(* IEC 61131-3 sources: codesys_template_public/codesys_export/Device/Application/Function Blocks/MC_BasicControl, 26 files *)

(* ---- MC_ActualDriver_SetPosition.st ---- *)
// X57s 驅動器不支援標準 MC_SetPosition（Set Position 指令）
// 使用 Homing Mode 35 模擬 SetPosition 的功能作為 Workaround
FUNCTION_BLOCK MC_ActualDriver_SetPosition
VAR_IN_OUT
	Axis : AXIS_REF_SM3;
END_VAR
VAR_INPUT
	Execute		: BOOL;
	Position	: LREAL;
	xReset		: BOOL;
END_VAR
VAR_OUTPUT
	Done	: BOOL;
	Busy	: BOOL;
	Error	: BOOL;
	ErrorID	: SM3_Basic.SMC_ERROR;
END_VAR
VAR
	iStep : INT;
	_fbMC_WriteHomingParameters : MC_WriteHomingParameters;
	_stFakeHomingParameter : structAxisControl_HomingProfile := (uiHomingMethod := 35);
	_fbMC_Home : MC_Home;
END_VAR

// === IMPLEMENTATION ===
_fbMC_WriteHomingParameters(Axis := Axis, xEnable := TRUE, stParameter := _stFakeHomingParameter);
_fbMC_Home(Axis := Axis, Position := Position);

CASE iStep OF
	0: // 等待 Execute
	_fbMC_WriteHomingParameters.xExecute := FALSE;
	_fbMC_Home.Execute := FALSE;
	Done := FALSE;
	Error := FALSE;
	Busy := FALSE;
	IF Execute THEN
		iStep := iStep + 1;
	END_IF

	1: // 寫入 Homing 參數（Homing Mode 35）
	_fbMC_WriteHomingParameters.xExecute := TRUE;
	Busy := TRUE;
	IF _fbMC_WriteHomingParameters.xDone THEN
		_fbMC_WriteHomingParameters.xExecute := FALSE;
		iStep := iStep + 1;
	END_IF
	IF _fbMC_WriteHomingParameters.xError THEN
		Error := TRUE;
		iStep := 9999;
	END_IF

	2: // 執行 MC_Home（使用 Mode 35 觸發位置設定）
	_fbMC_Home.Execute := TRUE;
	IF _fbMC_Home.Done THEN
		_fbMC_Home.Execute := FALSE;
		iStep := iStep + 1;
	END_IF
	IF _fbMC_Home.Error THEN
		Error := TRUE;
		ErrorID := _fbMC_Home.ErrorID;
		iStep := 9999;
	END_IF

ELSE // iStep >= 3 or 9999
	Done := (iStep <> 9999);
	IF NOT Execute THEN
		iStep := 0;
		Done := FALSE;
		Error := FALSE;
		ErrorID := 0;
	END_IF
END_CASE

IF xReset THEN
	iStep := 0;
	Done := FALSE;
	Error := FALSE;
	ErrorID := 0;
END_IF

(* ---- MC_BasicControl.st ---- *)
FUNCTION_BLOCK ABSTRACT MC_BasicControl EXTENDS BaseStateMachine
VAR_IN_OUT
	Axis        : AXIS_REF_SM3;
	stParameter : structAxisControl_Parameter;
END_VAR
VAR_INPUT
	xEMS         : BOOL;	// 緊急停止（立即，不等減速）
	xJogPositive : BOOL;	// Jog 正方向（跨任務持久訊號，HMI 用）
	xJogNegative : BOOL;	// Jog 負方向（跨任務持久訊號，HMI 用）
END_VAR
VAR_OUTPUT
	xAxisStandStill       : BOOL;	// 軸停止不動
	xPositiveLimitReached : BOOL;	// 正向極限觸動
	xNegativeLimitReached : BOOL;	// 負向極限觸動
	xInVelocity           : BOOL;	// 速度命令中（已達目標速度）
END_VAR
VAR
	// 電源控制旗標（由狀態機與 Stop() 管理）
	_xPowerOn : BOOL;

	// 驅動器 IO 旗標（由 ReadDriverInputs 填入）
	_xPositiveLimitInput : BOOL;
	_xNegativeLimitInput : BOOL;
	_xBrakeInput         : BOOL;
	_wDriverErrorCode    : WORD;

	// 命令請求旗標（當前掃描，由 method 設定）
	_xJogPosRequested  : BOOL;
	_xJogNegRequested  : BOOL;
	_xMoveAbsRequested : BOOL;
	_xMoveRelRequested : BOOL;
	_xMoveVelRequested : BOOL;
	_xHomeRequested    : BOOL;
	_xSetPosRequested  : BOOL;

	// 命令請求旗標（前一掃描，供狀態機讀取）
	_xJogPosRequested_Prev  : BOOL;
	_xJogNegRequested_Prev  : BOOL;
	_xMoveAbsRequested_Prev : BOOL;
	_xMoveRelRequested_Prev : BOOL;
	_xMoveVelRequested_Prev : BOOL;
	_xHomeRequested_Prev    : BOOL;
	_xSetPosRequested_Prev  : BOOL;

	// 命令參數（由 method 解析後填入）
	_lrJogVelocity : LREAL;
	_lrJogAcc      : LREAL;
	_lrJogDec      : LREAL;
	_lrJogJerk     : LREAL;

	_lrSetPosTarget : LREAL;

	// 命令完成追蹤
	_xCommandDone      : BOOL;
	_iActiveCommand    : INT;					// 最近完成的命令對應的 enumAxisControl_Step
	_eLastMotionError  : SM3_Error.SMC_ERROR;	// 最近一次 SM3 動作錯誤碼（供 method 回傳）

	// MoveRelative 重新觸發鎖：Done 後設 TRUE，呼叫端停止呼叫後清除
	// 防止持續呼叫 MoveRelative() 時完成後立刻開始下一次相對移動
	_xMoveRelNeedsReArm : BOOL;

	// 重置後返回步驟
	_iStepBeforeReset : INT;

	// SM3 Motion FBs
	_fbMC_Power                 : MC_Power;
	_fbMC_Reset                 : MC_Reset;
	_fbMC_MoveAbsolute          : MC_MoveAbsolute;
	_fbMC_MoveRelative          : MC_MoveRelative;
	_fbMC_MoveVelocity          : MC_MoveVelocity;
	_fbMC_Stop                  : MC_Stop;
	_fbMC_Stop_EMS              : MC_Stop;
	_fbMC_Home                  : MC_Home;
	_fbMC_WriteHomingParameters : MC_WriteHomingParameters;

	// Jog 速度變化偵測（ContinuousUpdate 邏輯）
	_fbVCD_Jog : ValueChangeDetector;
END_VAR

// === IMPLEMENTATION ===
xEnabled        := Axis.bRegulatorOn;
SUPER^();
_RunMotionFBs();

(* ---- MC_BasicControl_LC10E.st ---- *)
FUNCTION_BLOCK MC_BasicControl_LC10E EXTENDS MC_BasicControl
VAR_INPUT
	wDriverInputWord : WORD;	// X57s PDO 輸入字（位元映射見 ReadDriverInputs）
	wDriverErrorCode : WORD;	// X57s 錯誤碼（PDO 讀取）
END_VAR
VAR
	_fbSetPosition_ActualDriver : MC_ActualDriver_SetPosition;	// Homing Mode 35 workaround
	_xSetPosFirstCall   : BOOL := TRUE;			// 確保 Execute 有上升沿
END_VAR

// === IMPLEMENTATION ===
SUPER^(Axis := Axis, stParameter := stParameter);

(* ---- MC_BasicControl_VisuWrapper.st ---- *)
FUNCTION_BLOCK MC_BasicControl_VisuWrapper
VAR_IN_OUT
	fbAxis   : MC_BasicControl_LC10E;
	stCmd    : structMC_BasicControl_VisuCmd;
	stStatus : structMC_BasicControl_VisuStatus;
END_VAR
VAR
	_xClearLastResultPrev : BOOL;
	_xHomePrev            : BOOL;
	_xResetPrev           : BOOL;
	_xStopPrev            : BOOL;
	_xMoveAbsPrev         : BOOL;
	_xMoveRelPosPrev      : BOOL;
	_xMoveRelNegPrev      : BOOL;
	_xMoveVelPrev         : BOOL;
	_xSetPositionPrev     : BOOL;
	_xHomeLatched         : BOOL;
	_xMoveAbsLatched      : BOOL;
	_xMoveRelLatched      : BOOL;
	_xMoveVelLatched      : BOOL;
	_xSetPositionLatched  : BOOL;
	_udiLastPulseSeq   : UDINT;
END_VAR

// === IMPLEMENTATION ===
// Reject code:
// 1 = NONE command
// 2 = Unknown command
// 3 = Invalid motion parameter
stStatus.xPulseAccepted := FALSE;
stStatus.xPulseRejected := FALSE;
stStatus.iPulseRejectCode := 0;
stStatus.xJogCommanded := FALSE;

IF stCmd.xClearLastResult AND NOT _xClearLastResultPrev THEN
	Clear(stStatus.stLastResult);
END_IF

IF stCmd.xStop AND NOT _xStopPrev THEN
	fbAxis.Stop();
	_xHomeLatched := FALSE;
	_xMoveAbsLatched := FALSE;
	_xMoveRelLatched := FALSE;
	_xMoveVelLatched := FALSE;
	_xSetPositionLatched := FALSE;
	stStatus.xPulseAccepted := TRUE;
END_IF

IF stCmd.xReset AND NOT _xResetPrev THEN
	fbAxis.Reset();
	_xHomeLatched := FALSE;
	_xMoveAbsLatched := FALSE;
	_xMoveRelLatched := FALSE;
	_xMoveVelLatched := FALSE;
	_xSetPositionLatched := FALSE;
	stStatus.xPulseAccepted := TRUE;
END_IF

IF stCmd.udiPulseSeq <> _udiLastPulseSeq THEN
	CASE stCmd.ePulseCmd OF
		enumMC_BasicControl_VisuPulseCmd.STOP:
			fbAxis.Stop();
			_xHomeLatched := FALSE;
			_xMoveAbsLatched := FALSE;
			_xMoveRelLatched := FALSE;
			_xMoveVelLatched := FALSE;
			_xSetPositionLatched := FALSE;
			stStatus.xPulseAccepted := TRUE;
		enumMC_BasicControl_VisuPulseCmd.RESET:
			fbAxis.Reset();
			_xHomeLatched := FALSE;
			_xMoveAbsLatched := FALSE;
			_xMoveRelLatched := FALSE;
			_xMoveVelLatched := FALSE;
			_xSetPositionLatched := FALSE;
			stStatus.xPulseAccepted := TRUE;
		enumMC_BasicControl_VisuPulseCmd.HOME:
			_xHomeLatched := TRUE;
			_xMoveAbsLatched := FALSE;
			_xMoveRelLatched := FALSE;
			_xMoveVelLatched := FALSE;
			_xSetPositionLatched := FALSE;
			stStatus.xPulseAccepted := TRUE;
		enumMC_BasicControl_VisuPulseCmd.MOVE_ABSOLUTE:
			IF stCmd.lrMoveAbsVel < 0.0 OR stCmd.lrMoveAbsAcc < 0.0 OR stCmd.lrMoveAbsDec < 0.0 OR stCmd.lrMoveAbsJerk < 0.0 THEN
				stStatus.xPulseRejected := TRUE;
				stStatus.iPulseRejectCode := 3;
			ELSE
				_xHomeLatched := FALSE;
				_xMoveAbsLatched := TRUE;
				_xMoveRelLatched := FALSE;
				_xMoveVelLatched := FALSE;
				_xSetPositionLatched := FALSE;
				stStatus.xPulseAccepted := TRUE;
			END_IF
		enumMC_BasicControl_VisuPulseCmd.MOVE_RELATIVE:
			IF stCmd.lrMoveRelVel < 0.0 OR stCmd.lrMoveRelAcc < 0.0 OR stCmd.lrMoveRelDec < 0.0 OR stCmd.lrMoveRelJerk < 0.0 THEN
				stStatus.xPulseRejected := TRUE;
				stStatus.iPulseRejectCode := 3;
			ELSE
				_xHomeLatched := FALSE;
				_xMoveAbsLatched := FALSE;
				_xMoveRelLatched := TRUE;
				_xMoveVelLatched := FALSE;
				_xSetPositionLatched := FALSE;
				stStatus.xPulseAccepted := TRUE;
			END_IF
		enumMC_BasicControl_VisuPulseCmd.MOVE_VELOCITY:
			IF stCmd.lrMoveVelAcc < 0.0 OR stCmd.lrMoveVelDec < 0.0 OR stCmd.lrMoveVelJerk < 0.0 THEN
				stStatus.xPulseRejected := TRUE;
				stStatus.iPulseRejectCode := 3;
			ELSE
				_xHomeLatched := FALSE;
				_xMoveAbsLatched := FALSE;
				_xMoveRelLatched := FALSE;
				_xMoveVelLatched := TRUE;
				_xSetPositionLatched := FALSE;
				stStatus.xPulseAccepted := TRUE;
			END_IF
		enumMC_BasicControl_VisuPulseCmd.SET_POSITION:
			_xHomeLatched := FALSE;
			_xMoveAbsLatched := FALSE;
			_xMoveRelLatched := FALSE;
			_xMoveVelLatched := FALSE;
			_xSetPositionLatched := TRUE;
			stStatus.xPulseAccepted := TRUE;
		enumMC_BasicControl_VisuPulseCmd.NONE:
			stStatus.xPulseRejected := TRUE;
			stStatus.iPulseRejectCode := 1;
	ELSE
		stStatus.xPulseRejected := TRUE;
		stStatus.iPulseRejectCode := 2;
	END_CASE

	_udiLastPulseSeq      := stCmd.udiPulseSeq;
	stStatus.udiPulseAckSeq := stCmd.udiPulseSeq;
	stStatus.ePulseAckCmd   := stCmd.ePulseCmd;
END_IF

// Button pulse compatibility path for visu widgets.
IF stCmd.xHome AND NOT _xHomePrev THEN
	_xHomeLatched := TRUE;
	_xMoveAbsLatched := FALSE;
	_xMoveRelLatched := FALSE;
	_xMoveVelLatched := FALSE;
	_xSetPositionLatched := FALSE;
	stStatus.xPulseAccepted := TRUE;
ELSIF stCmd.xMoveAbsoluteExecute AND NOT _xMoveAbsPrev THEN
	IF stCmd.lrMoveAbsVel < 0.0 OR stCmd.lrMoveAbsAcc < 0.0 OR stCmd.lrMoveAbsDec < 0.0 OR stCmd.lrMoveAbsJerk < 0.0 THEN
		stStatus.xPulseRejected := TRUE;
		stStatus.iPulseRejectCode := 3;
	ELSE
		_xHomeLatched := FALSE;
		_xMoveAbsLatched := TRUE;
		_xMoveRelLatched := FALSE;
		_xMoveVelLatched := FALSE;
		_xSetPositionLatched := FALSE;
		stStatus.xPulseAccepted := TRUE;
	END_IF
ELSIF stCmd.xMoveRelativePosExecute AND NOT _xMoveRelPosPrev THEN
	IF stCmd.lrMoveRelVel < 0.0 OR stCmd.lrMoveRelAcc < 0.0 OR stCmd.lrMoveRelDec < 0.0 OR stCmd.lrMoveRelJerk < 0.0 THEN
		stStatus.xPulseRejected := TRUE;
		stStatus.iPulseRejectCode := 3;
	ELSE
		stCmd.lrMoveRelDist := ABS(stCmd.lrMoveRelDist);
		_xHomeLatched := FALSE;
		_xMoveAbsLatched := FALSE;
		_xMoveRelLatched := TRUE;
		_xMoveVelLatched := FALSE;
		_xSetPositionLatched := FALSE;
		stStatus.xPulseAccepted := TRUE;
	END_IF
ELSIF stCmd.xMoveRelativeNegExecute AND NOT _xMoveRelNegPrev THEN
	IF stCmd.lrMoveRelVel < 0.0 OR stCmd.lrMoveRelAcc < 0.0 OR stCmd.lrMoveRelDec < 0.0 OR stCmd.lrMoveRelJerk < 0.0 THEN
		stStatus.xPulseRejected := TRUE;
		stStatus.iPulseRejectCode := 3;
	ELSE
		stCmd.lrMoveRelDist := -ABS(stCmd.lrMoveRelDist);
		_xHomeLatched := FALSE;
		_xMoveAbsLatched := FALSE;
		_xMoveRelLatched := TRUE;
		_xMoveVelLatched := FALSE;
		_xSetPositionLatched := FALSE;
		stStatus.xPulseAccepted := TRUE;
	END_IF
ELSIF stCmd.xMoveVelocityExecute AND NOT _xMoveVelPrev THEN
	IF stCmd.lrMoveVelAcc < 0.0 OR stCmd.lrMoveVelDec < 0.0 OR stCmd.lrMoveVelJerk < 0.0 THEN
		stStatus.xPulseRejected := TRUE;
		stStatus.iPulseRejectCode := 3;
	ELSE
		_xHomeLatched := FALSE;
		_xMoveAbsLatched := FALSE;
		_xMoveRelLatched := FALSE;
		_xMoveVelLatched := TRUE;
		_xSetPositionLatched := FALSE;
		stStatus.xPulseAccepted := TRUE;
	END_IF
ELSIF stCmd.xSetPosition AND NOT _xSetPositionPrev THEN
	_xHomeLatched := FALSE;
	_xMoveAbsLatched := FALSE;
	_xMoveRelLatched := FALSE;
	_xMoveVelLatched := FALSE;
	_xSetPositionLatched := TRUE;
	stStatus.xPulseAccepted := TRUE;
END_IF

IF _xHomeLatched THEN
	stStatus.stLastResult := fbAxis.Home();
	IF stStatus.stLastResult.xDone OR stStatus.stLastResult.xError THEN
		_xHomeLatched := FALSE;
	END_IF
ELSIF _xMoveAbsLatched THEN
	stStatus.stLastResult := fbAxis.MoveAbsolute(
		lrPosition := stCmd.lrMoveAbsPos,
		lrVelocity := stCmd.lrMoveAbsVel,
		lrAcceleration := stCmd.lrMoveAbsAcc,
		lrDeceleration := stCmd.lrMoveAbsDec,
		lrJerk := stCmd.lrMoveAbsJerk
	);
	IF stStatus.stLastResult.xDone OR stStatus.stLastResult.xError THEN
		_xMoveAbsLatched := FALSE;
	END_IF
ELSIF _xMoveRelLatched THEN
	stStatus.stLastResult := fbAxis.MoveRelative(
		lrDistance := stCmd.lrMoveRelDist,
		lrVelocity := stCmd.lrMoveRelVel,
		lrAcceleration := stCmd.lrMoveRelAcc,
		lrDeceleration := stCmd.lrMoveRelDec,
		lrJerk := stCmd.lrMoveRelJerk
	);
	IF stStatus.stLastResult.xDone OR stStatus.stLastResult.xError THEN
		_xMoveRelLatched := FALSE;
	END_IF
ELSIF _xMoveVelLatched THEN
	stStatus.stLastResult := fbAxis.MoveVelocity(
		lrVelocity := stCmd.lrMoveVel,
		lrAcceleration := stCmd.lrMoveVelAcc,
		lrDeceleration := stCmd.lrMoveVelDec,
		lrJerk := stCmd.lrMoveVelJerk
	);
	IF stStatus.stLastResult.xError THEN
		_xMoveVelLatched := FALSE;
	END_IF
ELSIF _xSetPositionLatched THEN
	stStatus.stLastResult := fbAxis.SetPosition(lrPosition := stCmd.lrSetPosition);
	IF stStatus.stLastResult.xDone OR stStatus.stLastResult.xError THEN
		_xSetPositionLatched := FALSE;
	END_IF
END_IF

// Level command path (jog): hold TRUE to keep command active.
IF NOT (_xHomeLatched OR _xMoveAbsLatched OR _xMoveRelLatched OR _xMoveVelLatched OR _xSetPositionLatched) THEN
	IF stCmd.xJogPositive XOR stCmd.xJogNegative THEN
	IF stCmd.lrJogVelocity < 0.0 OR stCmd.lrJogAcc < 0.0 OR stCmd.lrJogDec < 0.0 OR stCmd.lrJogJerk < 0.0 THEN
		stStatus.xPulseRejected := TRUE;
		stStatus.iPulseRejectCode := 3;
	ELSIF stCmd.xJogPositive THEN
		stStatus.stLastResult := fbAxis.JogPositive(
			lrVelocity := stCmd.lrJogVelocity,
			lrAcceleration := stCmd.lrJogAcc,
			lrDeceleration := stCmd.lrJogDec,
			lrJerk := stCmd.lrJogJerk
		);
		stStatus.xJogCommanded := TRUE;
	ELSE
		stStatus.stLastResult := fbAxis.JogNegative(
			lrVelocity := stCmd.lrJogVelocity,
			lrAcceleration := stCmd.lrJogAcc,
			lrDeceleration := stCmd.lrJogDec,
			lrJerk := stCmd.lrJogJerk
		);
		stStatus.xJogCommanded := TRUE;
	END_IF
	END_IF
END_IF

IF stCmd.xRaiseDummyError THEN
	fbAxis.Raise(
		iErrorID:=enumAxisControl_ErrorID.DUMMY,
		iNextStep:=fbAxis.iStep
	);
END_IF

_xClearLastResultPrev := stCmd.xClearLastResult;
_xHomePrev := stCmd.xHome;
_xResetPrev := stCmd.xReset;
_xStopPrev := stCmd.xStop;
_xMoveAbsPrev := stCmd.xMoveAbsoluteExecute;
_xMoveRelPosPrev := stCmd.xMoveRelativePosExecute;
_xMoveRelNegPrev := stCmd.xMoveRelativeNegExecute;
_xMoveVelPrev := stCmd.xMoveVelocityExecute;
_xSetPositionPrev := stCmd.xSetPosition;

stStatus.xEnabled              := fbAxis.xEnabled;
stStatus.xBusy                 := fbAxis.xBusy;
stStatus.xDone                 := fbAxis.xDone;
stStatus.xError                := fbAxis.xError;
stStatus.iErrorID              := fbAxis.iErrorID;
stStatus.iStep                 := fbAxis.iStep;
stStatus.xAxisStandStill       := fbAxis.xAxisStandStill;
stStatus.xInVelocity           := fbAxis.xInVelocity;
stStatus.xInAcceleration       := FALSE;
stStatus.xInDeceleration       := FALSE;
stStatus.xPositiveLimitReached := fbAxis.xPositiveLimitReached;
stStatus.xNegativeLimitReached := fbAxis.xNegativeLimitReached;
stStatus.xBrakeSignal          := FALSE;

IF fbAxis.pAxis <> 0 THEN
	stStatus.lrActPosition := fbAxis.pAxis^.fActPosition;
	stStatus.lrActVelocity := fbAxis.pAxis^.fActVelocity;
	stStatus.lrSetPosition := fbAxis.pAxis^.fSetPosition;
	stStatus.lrSetVelocity := fbAxis.pAxis^.fSetVelocity;
END_IF

(* ---- MC_FuckTheDriver_SetPosition.st ---- *)
FUNCTION_BLOCK MC_FuckTheDriver_SetPosition
VAR_IN_OUT
	Axis : AXIS_REF_SM3;
END_VAR
VAR_INPUT
	Execute : BOOL;
	Position : LREAL;
	Mode : BOOL;
	xReset : BOOL;
END_VAR
VAR_OUTPUT
	Done : BOOL;
	Busy : BOOL;
	Error : BOOL;
	ErrorID : SM3_Basic.SMC_ERROR;
END_VAR
VAR
	iStep : INT;
	fbMC_WriteHomingParameters : MC_WriteHomingParameters;
	FakeHomingParameter : structAxisControl_HomingProfile :=
	(uiHomingMethod:=35);
	fbMC_Home : MC_Home;
END_VAR

// === IMPLEMENTATION ===
fbMC_WriteHomingParameters(Axis:=Axis,xEnable:=TRUE,stParameter:=FakeHomingParameter);
fbMC_Home(Axis:=Axis, Position:=Position);
CASE iStep OF
	0:
	fbMC_WriteHomingParameters.xExecute:=FALSE;
	fbMC_Home.Execute:=FALSE;
	IF Execute THEN
		iStep:=iStep+1;
	END_IF
	1:
	fbMC_WriteHomingParameters.xExecute:=TRUE;
	IF fbMC_WriteHomingParameters.xDone THEN
		fbMC_WriteHomingParameters.xExecute:=FALSE;
		iStep:=iStep+1;
	END_IF
	IF fbMC_WriteHomingParameters.xError THEN
		iStep:=9999;

	END_IF
	2:
	fbMC_Home.Execute:=TRUE;
	IF fbMC_Home.Done THEN
		fbMC_Home.Execute:=FALSE;
		iStep:=iStep+1;
	END_IF
	IF fbMC_Home.Error THEN
		iStep:=9999;
		Error:=TRUE;
		ErrorID:=fbMC_Home.ErrorID;
	END_IF
ELSE
	Done:=iStep<>9999;
	IF NOT Execute THEN
		iStep:=0;
		Done:=0;
		Error:=0;
		ErrorID:=0;
	END_IF
END_CASE
IF xReset THEN
	iStep:=0;
END_IF

(* ---- MC_IntegralPosition.st ---- *)
FUNCTION_BLOCK MC_IntegralPosition
VAR_IN_OUT
	Axis : AXIS_REF_SM3;
END_VAR
VAR_INPUT
	xEnable	: BOOL;
	xReset	: BOOL;

END_VAR
VAR_OUTPUT
	xBusy			: BOOL;
	lrCmdPosition	: LREAL;
	lrActPosition	: LREAL;
END_VAR
VAR
	lrScanTime	: LREAL;//sec
END_VAR

// === IMPLEMENTATION ===
IF xEnable THEN

	lrScanTime:=Axis.fTaskCycle;

	IF NOT xReset THEN
		lrCmdPosition:=lrCmdPosition+Axis.fSetVelocity*lrScanTime;
		lrActPosition:=lrActPosition+Axis.fActVelocity*lrScanTime;
	ELSE
		lrCmdPosition:=0;
		lrActPosition:=0;
	END_IF
END_IF

(* ---- MC_WriteHomingParameters.st ---- *)
FUNCTION_BLOCK MC_WriteHomingParameters EXTENDS BaseStateMachine
VAR_IN_OUT
	Axis 						: AXIS_REF_SM3;//指定軸
	stParameter					: structAxisControl_HomingProfile;//參數表
END_VAR

VAR_INPUT
END_VAR
VAR_OUTPUT
END_VAR
VAR CONSTANT
	//專用於寫入Homing參數的變數表
	//寫入順序:
	//1. Homing Acceleration
	//2. Speed during search for zero
	//3. Speed during search for switch
	//4. Homing method
	PARAMETER_SIZE : INT := 4;

	HOMING_PARAMETER_INDEXES : ARRAY [1..PARAMETER_SIZE] OF WORD :=
	[16#609A, 16#6099, 16#6099, 16#6098];

	HOMING_PARAMETER_SUBINDEXES : ARRAY [1..PARAMETER_SIZE] OF WORD :=
	[16#00, 16#02, 16#01, 16#00];

	HOMING_PARAMETER_SIZES : ARRAY [1..PARAMETER_SIZE] OF INT :=
	[4, 4, 4, 1];
END_VAR
VAR
	iWriteParameterIndex : INT;
	lrAryWriteParameterStack 	: ARRAY [1..PARAMETER_SIZE] OF LREAL;//寫入的棧數據
	fbMC_WriteParameter		: MC_WriteParameter;
	diParameterNumber : DINT;
END_VAR

// === IMPLEMENTATION ===
SUPER^();

(* ---- ValueChangeDetector.st ---- *)
FUNCTION_BLOCK ValueChangeDetector
VAR_INPUT
	In		: LREAL;
END_VAR
VAR_OUTPUT
	xValueChange_RisingTrig : BOOL;
END_VAR
VAR
	lrTemp : LREAL;
	rtValueChangeDetector : R_TRIG;
END_VAR

// === IMPLEMENTATION ===
rtValueChangeDetector(CLK:=In<>lrTemp,Q=>xValueChange_RisingTrig);
lrTemp:=In;

(* ---- MC_BasicControl._DetectErrors.st ---- *)
METHOD PRIVATE _DetectErrors

// === IMPLEMENTATION ===
// 偵測驅動器錯誤碼（已由 ReadDriverInputs 過濾已知正常碼）
// 觸發 Raise → 進入錯誤流程，TRY_RESET 後恢復
IF _wDriverErrorCode <> 0 THEN
	_ClearAllExecute();
	_eLastMotionError := THIS^._wDriverErrorCode;
	Raise(
		iErrorID  := enumAxisControl_ErrorID.DRIVER_ERROR,
		iNextStep := enumAxisControl_Step.TRY_RESET);
END_IF

(* ---- MC_BasicControl._RunMotionFBs.st ---- *)
METHOD PRIVATE _RunMotionFBs

// === IMPLEMENTATION ===
// 每掃描週期呼叫主要 SM3 FBs，避免命令狀態因間歇呼叫失步
// Execute 旗標由狀態機或 Stop() 控制

// MC_Power（_xPowerOn 由狀態機與 Stop() 管理）
_fbMC_Power(Axis := Axis, Enable := TRUE, bRegulatorOn := _xPowerOn, bDriveStart := _xPowerOn);

// MC_Reset（Execute 由 TRY_RESET/NOT_READY 控制）
_fbMC_Reset(Axis := Axis);

// 運動命令 FBs（Execute 由狀態機控制）
_fbMC_MoveAbsolute(Axis := Axis);
_fbMC_MoveRelative(Axis := Axis);
_fbMC_MoveVelocity(Axis := Axis);
_fbMC_Stop(Axis := Axis);
_fbMC_Home(Axis := Axis);

// WriteHomingParameters（僅在 homing 寫參數流程呼叫）
IF iStep = enumAxisControl_Step.HOMING_WRITE_PARAM OR
	_fbMC_WriteHomingParameters.xExecute THEN
	_fbMC_WriteHomingParameters(Axis := Axis, xEnable := TRUE, stParameter := stParameter.stHoming);
END_IF

// EMS 緊急停止（xEMS=TRUE 時立即停止，Jerk=0 表示最快減速）
_fbMC_Stop_EMS(Axis := Axis, Execute := xEMS, Deceleration := stParameter.lrEmergencyStopDec, Jerk := 0);

(* ---- MC_BasicControl.DoSetPosition.st ---- *)
METHOD ABSTRACT DoSetPosition : INT
VAR_INPUT
	lrPosition : LREAL;	// 目標位置
END_VAR
// 回傳值：
//   0 = 執行中（Busy）
//   1 = 完成（Done）
//  -1 = 錯誤（Error）
//
// 實作說明：子類需管理 Execute 邊緣偵測（上升沿觸發）
// 建議：使用內部旗標在首次呼叫時送出 Reset 脈衝

// === IMPLEMENTATION ===

(* ---- MC_BasicControl.InterrupMotionCommand.st ---- *)
METHOD PUBLIC InterrupMotionCommand : BOOL
VAR_INPUT
END_VAR

// === IMPLEMENTATION ===
iStep := enumAxisControl_Step.STOPPING;  // 中斷當前動作，進入停止序列
InterrupMotionCommand := TRUE;

(* ---- MC_BasicControl.JogNegative.st ---- *)
METHOD JogNegative : structAxisControl_Result
VAR_INPUT
	lrVelocity     : LREAL := 0;	// 0 = 使用 stParameter.stDefault.lrVelocity
	lrAcceleration : LREAL := 0;	// 0 = 使用 stParameter.stDefault.lrAcc
	lrDeceleration : LREAL := 0;	// 0 = 使用 stParameter.stDefault.lrDec
	lrJerk         : LREAL := 0;	// 0 = 使用 stParameter.stDefault.lrJerk
END_VAR

// === IMPLEMENTATION ===
_lrJogVelocity := SEL(lrVelocity     = 0, lrVelocity,     stParameter.stDefault.lrVelocity);
_lrJogAcc      := SEL(lrAcceleration = 0, lrAcceleration, stParameter.stDefault.lrAcc);
_lrJogDec      := SEL(lrDeceleration = 0, lrDeceleration, stParameter.stDefault.lrDec);
_lrJogJerk     := SEL(lrJerk         = 0, lrJerk,         stParameter.stDefault.lrJerk);

_fbMC_MoveVelocity.Velocity     := _lrJogVelocity;
_fbMC_MoveVelocity.Acceleration := _lrJogAcc;
_fbMC_MoveVelocity.Deceleration := _lrJogDec;
_fbMC_MoveVelocity.Jerk         := _lrJogJerk;

// 設定請求旗標（每掃描週期持續呼叫 = 持續 Jog）
_xJogNegRequested := TRUE;

// 回傳當前狀態
JogNegative.xBusy    := (iStep = enumAxisControl_Step.JOG_NEG);
JogNegative.xDone    := FALSE;	// Jog 沒有完成概念
JogNegative.xError   := xError;
JogNegative.eErrorID := _eLastMotionError;

(* ---- MC_BasicControl.JogPositive.st ---- *)
METHOD JogPositive : structAxisControl_Result
VAR_INPUT
	lrVelocity     : LREAL := 0;	// 0 = 使用 stParameter.stDefault.lrVelocity
	lrAcceleration : LREAL := 0;	// 0 = 使用 stParameter.stDefault.lrAcc
	lrDeceleration : LREAL := 0;	// 0 = 使用 stParameter.stDefault.lrDec
	lrJerk         : LREAL := 0;	// 0 = 使用 stParameter.stDefault.lrJerk
END_VAR

// === IMPLEMENTATION ===
_lrJogVelocity := SEL(lrVelocity     = 0, lrVelocity,     stParameter.stDefault.lrVelocity);
_lrJogAcc      := SEL(lrAcceleration = 0, lrAcceleration, stParameter.stDefault.lrAcc);
_lrJogDec      := SEL(lrDeceleration = 0, lrDeceleration, stParameter.stDefault.lrDec);
_lrJogJerk     := SEL(lrJerk         = 0, lrJerk,         stParameter.stDefault.lrJerk);

_fbMC_MoveVelocity.Velocity     := _lrJogVelocity;
_fbMC_MoveVelocity.Acceleration := _lrJogAcc;
_fbMC_MoveVelocity.Deceleration := _lrJogDec;
_fbMC_MoveVelocity.Jerk         := _lrJogJerk;

// 設定請求旗標（每掃描週期持續呼叫 = 持續 Jog）
_xJogPosRequested := TRUE;

// 回傳當前狀態
JogPositive.xBusy    := (iStep = enumAxisControl_Step.JOG_POS);
JogPositive.xDone    := FALSE;	// Jog 沒有完成概念
JogPositive.xError   := xError;
JogPositive.eErrorID := _eLastMotionError;

(* ---- MC_BasicControl.Main.st ---- *)
METHOD PROTECTED Main
VAR
	_iDoSetPosResult : INT;
END_VAR

// === IMPLEMENTATION ===
// ─── 1. 儲存並清除命令請求旗標 ────────────────────────────────────────────
// 將前一掃描週期 method 設定的旗標存入 _Prev，清除現旗標等待本週期重設
_ClearAndSaveRequestFlags();

// ─── 2. 讀取驅動器 IO（Abstract） ────────────────────────────────────────
// 子類填入 _xPositiveLimitInput, _xNegativeLimitInput, _xBrakeInput, _wDriverErrorCode
// 並更新 xPositiveLimitReached, xNegativeLimitReached
ReadDriverInputs();

// ─── 3. 更新輸出旗標 ──────────────────────────────────────────────────────
xAxisStandStill := Axis.nAxisState=SM3_Basic.SMC_AXIS_STATE.standstill;
xInVelocity     := Axis.bConstantVelocity;

// ─── 4. 偵測驅動器錯誤 ───────────────────────────────────────────────────
_DetectErrors();
IF xError THEN RETURN; END_IF

// ─── 5. 緊急停止（EMS） ──────────────────────────────────────────────────
// MC_Stop_EMS 已在 _RunMotionFBs() 中根據 xEMS 執行
// 此處負責清除其他命令並將狀態機移至安全狀態
IF xEMS THEN
	_ClearAllExecute();
	_fbMC_Stop.Execute := FALSE;
	IF iStep = enumAxisControl_Step.JOG_POS       OR
	   iStep = enumAxisControl_Step.JOG_NEG       OR
	   iStep = enumAxisControl_Step.MOVE_ABS      OR
	   iStep = enumAxisControl_Step.MOVE_REL      OR
	   iStep = enumAxisControl_Step.MOVE_VEL      OR
	   iStep = enumAxisControl_Step.HOMING_WRITE_PARAM OR
	   iStep = enumAxisControl_Step.HOMING_EXEC   OR
	   iStep = enumAxisControl_Step.SET_POSITION THEN
		iStep := enumAxisControl_Step.STOPPING;
	END_IF
	RETURN;
END_IF

// ─── 6. 狀態機 ────────────────────────────────────────────────────────────
CASE iStep OF

	// ── IDLE：等待 xEnable ──────────────────────────────────────────────
	enumAxisControl_Step.IDLE:
		_xPowerOn  := FALSE;
		xBusy      := FALSE;
		_xCommandDone := FALSE;
		IF xEnable THEN
			iStep := enumAxisControl_Step.ENABLING;
		END_IF

	// ── ENABLING：等待伺服使能完成 ─────────────────────────────────────
	enumAxisControl_Step.ENABLING:
		_xPowerOn := TRUE;
		xBusy     := TRUE;
		IF Axis.bRegulatorOn THEN
			iStep := enumAxisControl_Step.READY;
		ELSIF Axis.bError THEN
			iStep := enumAxisControl_Step.NOT_READY;
		END_IF

	// ── NOT_READY：軸有錯，嘗試 Reset 後再進入 READY ──────────────────
	enumAxisControl_Step.NOT_READY:
		_xPowerOn := TRUE;
		xBusy     := TRUE;
		_fbMC_Reset.Execute := TRUE;
		IF _fbMC_Reset.Done OR _fbMC_Reset.Error THEN
			_fbMC_Reset.Execute := FALSE;
		END_IF
		IF Axis.nAxisState=SM3_Basic.SMC_AXIS_STATE.standstill AND NOT Axis.bError THEN
			iStep := enumAxisControl_Step.READY;
		END_IF

	// ── READY：等待命令 ────────────────────────────────────────────────
	enumAxisControl_Step.READY:
		_xPowerOn     := TRUE;
		xBusy         := FALSE;
		_xCommandDone := FALSE;
		// MoveRelative 解鎖：呼叫端停止呼叫時清除重觸旗標
		IF NOT _xMoveRelRequested_Prev THEN
			_xMoveRelNeedsReArm := FALSE;
		END_IF
		// 命令分派（優先順序由上而下）
		IF _xMoveAbsRequested_Prev THEN
			iStep := enumAxisControl_Step.MOVE_ABS;
		ELSIF _xMoveRelRequested_Prev AND NOT _xMoveRelNeedsReArm THEN
			iStep := enumAxisControl_Step.MOVE_REL;
		ELSIF _xMoveVelRequested_Prev THEN
			iStep := enumAxisControl_Step.MOVE_VEL;
		ELSIF (_xJogPosRequested_Prev OR xJogPositive) AND NOT _xPositiveLimitInput THEN
			iStep := enumAxisControl_Step.JOG_POS;
		ELSIF (_xJogNegRequested_Prev OR xJogNegative) AND NOT _xNegativeLimitInput THEN
			iStep := enumAxisControl_Step.JOG_NEG;
		ELSIF _xHomeRequested_Prev THEN
			iStep := enumAxisControl_Step.HOMING_WRITE_PARAM;
		ELSIF _xSetPosRequested_Prev THEN
			iStep := enumAxisControl_Step.SET_POSITION;
		END_IF

	// ── JOG_POS：正方向點動 ────────────────────────────────────────────
	enumAxisControl_Step.JOG_POS:
		xBusy := TRUE;
		_fbMC_MoveVelocity.Direction	:= SM3_Basic.MC_DIRECTION.positive;
		// ContinuousUpdate 模式：TRUE=持續刷新 Execute；FALSE=速度變化時重啟
		IF stParameter.xContinuousUpdate THEN
			_fbMC_MoveVelocity.Execute := TRUE;
		ELSE
			_fbVCD_Jog(In := _lrJogVelocity);
			IF _fbVCD_Jog.xValueChange_RisingTrig THEN
				_fbMC_MoveVelocity.Execute := FALSE;	// 短暫降低，下一掃描重啟
			ELSE
				_fbMC_MoveVelocity.Execute := TRUE;
			END_IF
		END_IF
		// 正向極限觸動：停止並嘗試重置
		IF _xPositiveLimitInput THEN
			_fbMC_MoveVelocity.Execute := FALSE;
			Raise(iErrorID  := enumAxisControl_ErrorID.POSITIVE_LIMIT_TRIP,
			      iNextStep := enumAxisControl_Step.TRY_RESET);
			RETURN;
		END_IF
		// 命令取消（method 停止呼叫）
		IF NOT (_xJogPosRequested_Prev OR xJogPositive) THEN
			_fbMC_MoveVelocity.Execute := FALSE;
			iStep := enumAxisControl_Step.STOPPING;
		END_IF
		IF _fbMC_MoveVelocity.Error THEN
			_fbMC_MoveVelocity.Execute := FALSE;
			_eLastMotionError := _fbMC_MoveVelocity.ErrorID;
			Raise(iErrorID  := enumAxisControl_ErrorID.DRIVER_ERROR,
			      iNextStep := enumAxisControl_Step.TRY_RESET);
			RETURN;
		END_IF

	// ── JOG_NEG：負方向點動 ────────────────────────────────────────────
	enumAxisControl_Step.JOG_NEG:
		xBusy := TRUE;
		_fbMC_MoveVelocity.Direction	:= SM3_Basic.MC_DIRECTION.negative;
		// ContinuousUpdate 邏輯（追蹤絕對速度值）
		IF stParameter.xContinuousUpdate THEN
			_fbMC_MoveVelocity.Execute := TRUE;
		ELSE
			_fbVCD_Jog(In := _lrJogVelocity);
			IF _fbVCD_Jog.xValueChange_RisingTrig THEN
				_fbMC_MoveVelocity.Execute := FALSE;
			ELSE
				_fbMC_MoveVelocity.Execute := TRUE;
			END_IF
		END_IF
		// 負向極限觸動
		IF _xNegativeLimitInput THEN
			_fbMC_MoveVelocity.Execute := FALSE;
			Raise(iErrorID  := enumAxisControl_ErrorID.NEGATIVE_LIMIT_TRIP,
			      iNextStep := enumAxisControl_Step.TRY_RESET);
			RETURN;
		END_IF
		// 命令取消
		IF NOT (_xJogNegRequested_Prev OR xJogNegative) THEN
			_fbMC_MoveVelocity.Execute := FALSE;
			iStep := enumAxisControl_Step.STOPPING;
		END_IF
		IF _fbMC_MoveVelocity.Error THEN
			_fbMC_MoveVelocity.Execute := FALSE;
			_eLastMotionError := _fbMC_MoveVelocity.ErrorID;
			Raise(iErrorID  := enumAxisControl_ErrorID.DRIVER_ERROR,
			      iNextStep := enumAxisControl_Step.TRY_RESET);
			RETURN;
		END_IF

	// ── MOVE_ABS：絕對位置移動 ────────────────────────────────────────
	enumAxisControl_Step.MOVE_ABS:
		xBusy := TRUE;
		_fbMC_MoveAbsolute.Execute      := TRUE;
		IF _fbMC_MoveAbsolute.Done THEN
			_xCommandDone   := TRUE;
			_iActiveCommand := enumAxisControl_Step.MOVE_ABS;
			_ClearAllExecute();
			iStep := enumAxisControl_Step.STOPPING;
		ELSIF _fbMC_MoveAbsolute.Error THEN
			_ClearAllExecute();
			_eLastMotionError := _fbMC_MoveAbsolute.ErrorID;
			Raise(iErrorID  := enumAxisControl_ErrorID.MOVE_ABS_FAIL,
			      iNextStep := enumAxisControl_Step.READY);
			RETURN;
		ELSIF NOT _xMoveAbsRequested_Prev THEN
			// 呼叫端停止呼叫 MoveAbsolute() → 取消
			_ClearAllExecute();
			iStep := enumAxisControl_Step.STOPPING;
		END_IF

	// ── MOVE_REL：相對位置移動 ────────────────────────────────────────
	enumAxisControl_Step.MOVE_REL:
		xBusy := TRUE;
		_fbMC_MoveRelative.Execute      := TRUE;
		IF _fbMC_MoveRelative.Done THEN
			_xCommandDone       := TRUE;
			_iActiveCommand     := enumAxisControl_Step.MOVE_REL;
			_xMoveRelNeedsReArm := TRUE;	// 鎖住：防止呼叫端持續呼叫時立刻重新執行
			_ClearAllExecute();
			iStep := enumAxisControl_Step.STOPPING;
		ELSIF _fbMC_MoveRelative.Error THEN
			_ClearAllExecute();
			_eLastMotionError := _fbMC_MoveRelative.ErrorID;
			Raise(iErrorID  := enumAxisControl_ErrorID.MOVE_REL_FAIL,
			      iNextStep := enumAxisControl_Step.READY);
			RETURN;
		ELSIF NOT _xMoveRelRequested_Prev THEN
			_ClearAllExecute();
			iStep := enumAxisControl_Step.STOPPING;
		END_IF

	// ── MOVE_VEL：速度模式（持續）───────────────────────────────────
	enumAxisControl_Step.MOVE_VEL:
		xBusy := TRUE;
		_fbMC_MoveVelocity.Execute      := TRUE;
		IF _fbMC_MoveVelocity.Error THEN
			_ClearAllExecute();
			_eLastMotionError := _fbMC_MoveVelocity.ErrorID;
			Raise(iErrorID  := enumAxisControl_ErrorID.MOVE_VEL_FAIL,
			      iNextStep := enumAxisControl_Step.READY);
			RETURN;
		ELSIF NOT _xMoveVelRequested_Prev THEN
			// 呼叫端停止呼叫 MoveVelocity() → 停止
			_fbMC_MoveVelocity.Execute := FALSE;
			iStep := enumAxisControl_Step.STOPPING;
		END_IF

	// ── HOMING_WRITE_PARAM：寫入回原點驅動器參數 ─────────────────────
	enumAxisControl_Step.HOMING_WRITE_PARAM:
		xBusy := TRUE;
		_fbMC_WriteHomingParameters.xExecute := TRUE;
		IF _fbMC_WriteHomingParameters.xDone THEN
			_fbMC_WriteHomingParameters.xExecute := FALSE;
			iStep := enumAxisControl_Step.HOMING_EXEC;
		ELSIF _fbMC_WriteHomingParameters.xError THEN
			_ClearAllExecute();
			_eLastMotionError := _fbMC_WriteHomingParameters.iErrorID;
			Raise(iErrorID  := enumAxisControl_ErrorID.HOMING_WRITE_PARAM_FAIL,
			      iNextStep := enumAxisControl_Step.READY);
			RETURN;
		ELSIF NOT _xHomeRequested_Prev THEN
			_ClearAllExecute();
			iStep := enumAxisControl_Step.STOPPING;
		END_IF

	// ── HOMING_EXEC：執行回原點動作 ───────────────────────────────────
	enumAxisControl_Step.HOMING_EXEC:
		xBusy := TRUE;
		_fbMC_Home.Position := stParameter.stHoming.lrHomingPositionOffset;
		_fbMC_Home.Execute  := TRUE;
		IF _fbMC_Home.Done THEN
			_xCommandDone   := TRUE;
			_iActiveCommand := enumAxisControl_Step.HOMING_EXEC;
			_ClearAllExecute();
			iStep := enumAxisControl_Step.STOPPING;
		ELSIF _fbMC_Home.Error THEN
			_ClearAllExecute();
			_eLastMotionError := _fbMC_Home.ErrorID;
			Raise(iErrorID  := enumAxisControl_ErrorID.HOMING_EXEC_FAIL,
			      iNextStep := enumAxisControl_Step.READY);
			RETURN;
		ELSIF NOT _xHomeRequested_Prev THEN
			_ClearAllExecute();
			iStep := enumAxisControl_Step.STOPPING;
		END_IF

	// ── SET_POSITION：設定座標（不含運動）───────────────────────────
	enumAxisControl_Step.SET_POSITION:
		xBusy := TRUE;
		// DoSetPosition 為 Abstract，由子類實作（管理 Execute 邊緣邏輯）
		_iDoSetPosResult := DoSetPosition(lrPosition := _lrSetPosTarget);
		IF _iDoSetPosResult = 1 THEN
			_xCommandDone   := TRUE;
			_iActiveCommand := enumAxisControl_Step.SET_POSITION;
			// SetPosition 不涉及運動，完成後直接回 READY
			iStep := enumAxisControl_Step.READY;
		ELSIF _iDoSetPosResult = -1 THEN
			Raise(iErrorID  := enumAxisControl_ErrorID.SET_POSITION_FAIL,
			      iNextStep := enumAxisControl_Step.READY);
			RETURN;
		END_IF

	// ── STOPPING：觸發 MC_Stop，立即進入 WAIT_STOP ───────────────────
	enumAxisControl_Step.STOPPING:
		xBusy := TRUE;
		IF NOT xEMS THEN
			// EMS 時改用 MC_Stop_EMS，不重複啟動 MC_Stop
			_fbMC_Stop.Deceleration := stParameter.lrStopDec;
			_fbMC_Stop.Jerk         := stParameter.lrStopJerk;
			_fbMC_Stop.Execute      := TRUE;
		END_IF
		iStep := enumAxisControl_Step.WAIT_STOP;

	// ── WAIT_STOP：等待停止完成 ────────────────────────────────────────
	enumAxisControl_Step.WAIT_STOP:
		xBusy := TRUE;
		IF xEMS THEN
			// EMS 時等待軸實際靜止（由 MC_Stop_EMS 控制）
			IF Axis.nAxisState=SM3_Basic.SMC_AXIS_STATE.standstill AND NOT xStop THEN
				iStep := enumAxisControl_Step.READY;
			END_IF
		ELSE
			IF _fbMC_Stop.Done AND NOT xStop THEN
				_xCommandDone   := TRUE;
				_iActiveCommand := enumAxisControl_Step.STOPPING;
				_fbMC_Stop.Execute := FALSE;
				iStep := enumAxisControl_Step.READY;
			END_IF
			IF _fbMC_Stop.Error THEN
				_fbMC_Stop.Execute := FALSE;
				_eLastMotionError := _fbMC_Stop.ErrorID;
				Raise(iErrorID  := enumAxisControl_ErrorID.DRIVER_ERROR,
				      iNextStep := enumAxisControl_Step.TRY_RESET);
				RETURN;
			END_IF
		END_IF

	// ── TRY_RESET：驅動器重置後恢復 ────────────────────────────────
	enumAxisControl_Step.TRY_RESET:
		xBusy := TRUE;
		_fbMC_Reset.Execute := TRUE;
		IF _fbMC_Reset.Done OR _fbMC_Reset.ErrorID=SM3_Error.SMC_R_NO_ERROR_TO_RESET THEN
			_fbMC_Reset.Execute := FALSE;
			IF Axis.nAxisState=SM3_Basic.SMC_AXIS_STATE.standstill AND NOT Axis.bError THEN
				iStep := _iStepBeforeReset;
			END_IF
		END_IF
		IF _fbMC_Reset.Error THEN
			_fbMC_Reset.Execute := FALSE;
			// 重置失敗：停留在 TRY_RESET 等待外部干預（xReset）
		END_IF

END_CASE

(* ---- MC_BasicControl.MoveAbsolute.st ---- *)
METHOD MoveAbsolute : structAxisControl_Result
VAR_INPUT
	lrPosition     : LREAL;		// 目標絕對位置（必填）
	lrVelocity     : LREAL := 0;	// 0 = 使用 stParameter.stDefault.lrVelocity
	lrAcceleration : LREAL := 0;	// 0 = 使用 stParameter.stDefault.lrAcc
	lrDeceleration : LREAL := 0;	// 0 = 使用 stParameter.stDefault.lrDec
	lrJerk         : LREAL := 0;	// 0 = 使用 stParameter.stDefault.lrJerk
END_VAR

// === IMPLEMENTATION ===
// 解析有效參數（0 = 使用預設）
_fbMC_MoveAbsolute.Position     := lrPosition;
_fbMC_MoveAbsolute.Velocity     := SEL(lrVelocity     = 0, lrVelocity,     stParameter.stDefault.lrVelocity);
_fbMC_MoveAbsolute.Acceleration := SEL(lrAcceleration = 0, lrAcceleration, stParameter.stDefault.lrAcc);
_fbMC_MoveAbsolute.Deceleration := SEL(lrDeceleration = 0, lrDeceleration, stParameter.stDefault.lrDec);
_fbMC_MoveAbsolute.Jerk         := SEL(lrJerk         = 0, lrJerk,         stParameter.stDefault.lrJerk);

// 設定請求旗標（下一掃描週期 FB body 讀取 _Prev 版本）
_xMoveAbsRequested := TRUE;

// 回傳當前狀態
MoveAbsolute.xBusy  := (iStep = enumAxisControl_Step.MOVE_ABS);
MoveAbsolute.xDone  := _xCommandDone AND (_iActiveCommand = enumAxisControl_Step.MOVE_ABS);
MoveAbsolute.xError := xError;
MoveAbsolute.eErrorID := _eLastMotionError;

(* ---- MC_BasicControl.MoveRelative.st ---- *)
METHOD MoveRelative : structAxisControl_Result
VAR_INPUT
	lrDistance     : LREAL;		// 移動距離（正值=正方向，負值=負方向）
	lrVelocity     : LREAL := 0;	// 0 = 使用 stParameter.stDefault.lrVelocity
	lrAcceleration : LREAL := 0;	// 0 = 使用 stParameter.stDefault.lrAcc
	lrDeceleration : LREAL := 0;	// 0 = 使用 stParameter.stDefault.lrDec
	lrJerk         : LREAL := 0;	// 0 = 使用 stParameter.stDefault.lrJerk
END_VAR

// === IMPLEMENTATION ===
// 解析有效參數（0 = 使用預設）
_fbMC_MoveRelative.Distance     := lrDistance;
_fbMC_MoveRelative.Velocity     := SEL(lrVelocity     = 0, lrVelocity,     stParameter.stDefault.lrVelocity);
_fbMC_MoveRelative.Acceleration := SEL(lrAcceleration = 0, lrAcceleration, stParameter.stDefault.lrAcc);
_fbMC_MoveRelative.Deceleration := SEL(lrDeceleration = 0, lrDeceleration, stParameter.stDefault.lrDec);
_fbMC_MoveRelative.Jerk         := SEL(lrJerk         = 0, lrJerk,         stParameter.stDefault.lrJerk);

// 設定請求旗標
_xMoveRelRequested := TRUE;

// 回傳當前狀態
MoveRelative.xBusy    := (iStep = enumAxisControl_Step.MOVE_REL);
MoveRelative.xDone    := _xCommandDone AND (_iActiveCommand = enumAxisControl_Step.MOVE_REL);
MoveRelative.xError   := xError;
MoveRelative.eErrorID := _eLastMotionError;

(* ---- MC_BasicControl.MoveVelocity.st ---- *)
METHOD MoveVelocity : structAxisControl_Result
VAR_INPUT
	lrVelocity     : LREAL := 0;	// 速度（正=正向，負=負向），0 使用預設
	lrAcceleration : LREAL := 0;	// 0 = 使用 stParameter.stDefault.lrAcc
	lrDeceleration : LREAL := 0;	// 0 = 使用 stParameter.stDefault.lrDec
	lrJerk         : LREAL := 0;	// 0 = 使用 stParameter.stDefault.lrJerk
END_VAR

// === IMPLEMENTATION ===
_fbMC_MoveVelocity.Velocity     := SEL(lrVelocity     = 0, lrVelocity,     stParameter.stDefault.lrVelocity);
_fbMC_MoveVelocity.Acceleration := SEL(lrAcceleration = 0, lrAcceleration, stParameter.stDefault.lrAcc);
_fbMC_MoveVelocity.Deceleration := SEL(lrDeceleration = 0, lrDeceleration, stParameter.stDefault.lrDec);
_fbMC_MoveVelocity.Jerk         := SEL(lrJerk         = 0, lrJerk,         stParameter.stDefault.lrJerk);

// 設定請求旗標
_xMoveVelRequested := TRUE;

// 回傳當前狀態（MoveVelocity 沒有 xDone，只有 xBusy = InVelocity）
MoveVelocity.xBusy    := (iStep = enumAxisControl_Step.MOVE_VEL);
MoveVelocity.xDone    := FALSE;
MoveVelocity.xError   := xError;
MoveVelocity.eErrorID := _eLastMotionError;

(* ---- MC_BasicControl.pAxis.st ---- *)
PROPERTY pAxis : POINTER TO AXIS_REF_SM3

// === IMPLEMENTATION ===
// === GET ===
VAR
END_VAR

// === IMPLEMENTATION ===
pAxis:=ADR(THIS^.Axis);

(* ---- MC_BasicControl.pParameter.st ---- *)
PROPERTY pParameter : POINTER TO structAxisControl_Parameter

// === IMPLEMENTATION ===
// === GET ===
VAR
END_VAR

// === IMPLEMENTATION ===
pParameter:=ADR(THIS^.stParameter);

(* ---- MC_BasicControl.Reset.st ---- *)
METHOD Reset : BOOL

// === IMPLEMENTATION ===
// 覆蓋 BaseStateMachine.Reset()：
// 不恢復 iLastStep，而是進入 TRY_RESET 讓驅動器確實重置後再恢復 READY
IF xError THEN
	_ClearAllExecute();
	_fbMC_Stop.Execute  := FALSE;
	_fbMC_Reset.Execute := FALSE;
	iStep               := enumAxisControl_Step.TRY_RESET;
	_iStepBeforeReset   := enumAxisControl_Step.READY;
	xError              := FALSE;
	iErrorID            := 0;
	Reset               := TRUE;
END_IF
// 不呼叫 SUPER^.Reset()

(* ---- MC_BasicControl.SetPosition.st ---- *)
METHOD SetPosition : structAxisControl_Result
VAR_INPUT
	lrPosition : LREAL;		// 目標位置設定值
END_VAR

// === IMPLEMENTATION ===
_lrSetPosTarget   := lrPosition;
_xSetPosRequested := TRUE;

// 回傳當前狀態
SetPosition.xBusy    := (iStep = enumAxisControl_Step.SET_POSITION);
SetPosition.xDone    := _xCommandDone AND (_iActiveCommand = enumAxisControl_Step.SET_POSITION);
SetPosition.xError   := xError;
SetPosition.eErrorID := _eLastMotionError;

(* ---- MC_BasicControl.StopMotion.st ---- *)
METHOD StopMotion : structAxisControl_Result

// === IMPLEMENTATION ===
// 區分兩種 Stop 場景：
// - xEnable=FALSE：完全斷電，回到 IDLE（iStep=0）
// - xStop=TRUE：  停止運動，保持供電（狀態機繼續管理）
IF NOT xEnable THEN
	_xPowerOn := FALSE;
	_ClearAllExecute();
	_fbMC_Stop.Execute := FALSE;
	SUPER^.Stop();	// iStep := 0, xBusy/xDone/xError := FALSE
ELSE
	// xStop=TRUE 場景：只在不已處於停止流程時才轉換
	IF iStep <> enumAxisControl_Step.STOPPING AND
	   iStep <> enumAxisControl_Step.WAIT_STOP THEN
		_ClearAllExecute();
		iStep := enumAxisControl_Step.STOPPING;
	END_IF
END_IF

// 回傳當前狀態
StopMotion.xBusy := (iStep = enumAxisControl_Step.STOPPING OR iStep = enumAxisControl_Step.WAIT_STOP);
StopMotion.xDone := _xCommandDone AND (_iActiveCommand = enumAxisControl_Step.STOPPING);
StopMotion.xError := xError;
StopMotion.eErrorID := _eLastMotionError;

(* ---- MC_BasicControl_LC10E.DoSetPosition.st ---- *)
METHOD DoSetPosition : INT
VAR_INPUT
	lrPosition : LREAL;
END_VAR

// === IMPLEMENTATION ===
// X57s 不支援標準 MC_SetPosition，使用 Homing Mode 35 作為 workaround
// _xSetPosFirstCall 確保每次進入 SET_POSITION 狀態時有 Execute 上升沿

IF _xSetPosFirstCall THEN
	// 首次呼叫：送出 Reset 脈衝，確保 FB 從乾淨狀態開始
	_fbSetPosition_ActualDriver(Axis := Axis, Execute := FALSE, Position := lrPosition, xReset := TRUE);
	_xSetPosFirstCall := FALSE;
ELSE
	_fbSetPosition_ActualDriver(Axis := Axis, Execute := TRUE, Position := lrPosition, xReset := FALSE);
END_IF

IF _fbSetPosition_ActualDriver.Done THEN
	_xSetPosFirstCall := TRUE;		// 重置，供下次使用
	DoSetPosition := 1;
ELSIF _fbSetPosition_ActualDriver.Error THEN
	_xSetPosFirstCall := TRUE;
	DoSetPosition := -1;
ELSE
	DoSetPosition := 0;
END_IF

(* ---- MC_BasicControl_LC10E.ReadDriverInputs.st ---- *)
METHOD ReadDriverInputs
VAR
	_wFilteredCode : WORD;
END_VAR

// === IMPLEMENTATION ===
// 過濾 X57s 已知的正常狀態碼（非真實錯誤）
_wFilteredCode := wDriverErrorCode;
IF _wFilteredCode=21571 THEN//正極限
	_wFilteredCode:=0;
END_IF
IF _wFilteredCode=21572 THEN//負極限
	_wFilteredCode:=0;
END_IF

_wDriverErrorCode := _wFilteredCode;

// wDriverInputWord 位元映射（X57s PDO 定義）
_xPositiveLimitInput := wDriverInputWord.0;
_xNegativeLimitInput := wDriverInputWord.1;
_xBrakeInput         := wDriverInputWord.2;

// 更新輸出旗標
xPositiveLimitReached := _xPositiveLimitInput;
xNegativeLimitReached := _xNegativeLimitInput;

(* ---- MC_WriteHomingParameters.Main.st ---- *)
METHOD PROTECTED Main
VAR
	i : INT;
END_VAR

// === IMPLEMENTATION ===
CASE THIS^.iStep OF
	0://Init
	xBusy:=0;
	xError:=0;
	iErrorID:=0;
	fbMC_WriteParameter.Execute:=0;
	iWriteParameterIndex:=0;
	IF xExecute THEN
		iStep:=iStep+1;
	END_IF
	1:
	IF NOT fbMC_WriteParameter.Busy THEN
		iStep:=iStep+1;
		xBusy:=1;
	END_IF
	2:
	//處理數據
	lrAryWriteParameterStack[1]:=
		stParameter.lrHoming_Acceleration*
		stParameter.lrUnitToPulseRatio;
	lrAryWriteParameterStack[2]:=
		stParameter.lrVelocityDuringSearchForZero*
		stParameter.lrUnitToPulseRatio;
	lrAryWriteParameterStack[3]:=
		stParameter.lrVelocityDuringSearchForSwitch*
		stParameter.lrUnitToPulseRatio;
	lrAryWriteParameterStack[4]:=
		stParameter.uiHomingMethod;
	FOR i:=1 TO PARAMETER_SIZE DO
		IF lrAryWriteParameterStack[i]=SM3_Math.SMC_Math_Global.NaN THEN
			iStep:=9999;
			xError:=1;
		END_IF
	END_FOR
	iWriteParameterIndex:=1;
	iStep:=iStep+1;
	3:
	//寫入數據
	//這是說明書有關MC_WriteParameter上的公式，別動
	diParameterNumber :=
	- DWORD_TO_DINT(
		SHL(TO_DWORD(HOMING_PARAMETER_SIZES[iWriteParameterIndex]), 24)+
		SHL(TO_DWORD(HOMING_PARAMETER_INDEXES[iWriteParameterIndex]), 8)+
		HOMING_PARAMETER_SUBINDEXES[iWriteParameterIndex]
		);
	//指定參數
	fbMC_WriteParameter.ParameterNumber:=diParameterNumber;
	fbMC_WriteParameter.Value:=lrAryWriteParameterStack[iWriteParameterIndex];
	fbMC_WriteParameter.Execute:=1;
	iStep:=iStep+1;
	4:
	IF fbMC_WriteParameter.Done THEN//寫入完成
		fbMC_WriteParameter.Execute:=0;
		iWriteParameterIndex:=iWriteParameterIndex+1;
		IF iWriteParameterIndex>PARAMETER_SIZE THEN//若參數全部寫入完成則退出
			iStep:=100;
		ELSE//參數還沒全部寫入完成，則退到上一步繼續寫入
			iStep:=iStep-1;
		END_IF
	END_IF
	IF fbMC_WriteParameter.Error THEN
	 xError:=TRUE;
	 iErrorID:=fbMC_WriteParameter.ErrorID;
	 iStep:=9999;
	END_IF
ELSE
	xDone:=1;
	IF NOT xExecute THEN
		xDone:=0;
		iStep:=0;
	END_IF
END_CASE
fbMC_WriteParameter(Axis:=Axis);
